# EPICS autosave request: eigerApp/Db/eiger1_settings.req
file "eigerBase_settings.req", P=$(P), R=$(R)
